Fanuc KAREL source: ko00058.KL

PROGRAM KO00058
%STACKSIZE=65535
%PRIORITY=65535
%NOLOCKGROUP
VAR
P1 : XYZWPR
P2 : XYZWPREXT
F : BOOLEAN
OUT : XYZWPR
BEGIN
F=TRUE
-- UNSAFE_SOURCE_IR line 11: OUT = MIRROR(convert_xyzwpr_to_xyzwprext(P1), convert_xyzwprext_to_position(P2), F)
END KO00058
